(*
SPDX-FileCopyrightText: Â© 2026 Oleksandr Tiutyk <trofimich@gmail.com>
SPDX-License-Identifier: MIT
License: https://opensource.org/license/mit
*)

(*!
<summary>Base leaf automation component providing cyclic input processing.</summary>
<description>
Derived components override OnProcessInput to read inputs from hardware or communications.
ProcessInput executes the hook within a guarded TRY/CATCH block.
</description>
*)

FUNCTION_BLOCK ABSTRACT InputLeafAutomationComponent EXTENDS LeafAutomationComponent
	IMPLEMENTS IInputLeafAutomationComponent

(*!
<summary>Override to perform cyclic reading of input data.</summary>
*)
METHOD PROTECTED ABSTRACT OnProcessInput
END_METHOD

(*!
<summary>Invokes OnProcessInput with standardized exception handling and error dispatching.</summary>
*)
METHOD FINAL ProcessInput
VAR
	exceptionCode : __SYSTEM.ExceptionCode;
	exception : TOF_Core.IException;
	exceptionReaction : TOF_Core.EXCEPTION_REACTION;
END_VAR
__TRY
	OnProcessInput();
__CATCH(exceptionCode)		
	exception := TOF_Core.ExceptionManager.GetLastException(
		exceptionCode := exceptionCode,
		catchPointNamespaceName := NamespaceName,
		catchPointPOUName := __POUNAME(),
		catchPointPosition := __POSITION()
	);
					
	exceptionReaction := OnHandleException(exception := exception, failedMethodName := 'OnProcessInput');

	ProcessException(
		exception := exception,
		exceptionReaction := exceptionReaction,
		exceptionSourceHint := "OnProcessInput error"
	);
__ENDTRY
END_METHOD

END_FUNCTION_BLOCK

(* stored: Version 1.1.0.1
   POU InputLeafAutomationComponent: Id {efa8b231-2751-492d-8626-738af2170475}, SpecialFunc None
   Folder Methods to override: Id {57e5027c-d025-4d1f-bcea-3cc2ecc52027}
   Method OnProcessInput: Id {30690d44-71d9-48d1-97f7-67db91fa17cb}
   Method ProcessInput: Id {c8983ed6-ea33-4eb7-a3f3-5a36dc5ceb9e} *)
